PROGRAM MAIN
VAR
END_VAR

END_PROGRAM

(* stored: Version 1.1.0.1
   POU MAIN: Id {7bade889-ff3b-4ca4-b6fc-00ee581b029c} *)
